Staubli VAL3: JTrajPtFullBody.dtx

public num accelerations[10]
public num positions[10]
public num robotId
public num sequence
public num time
public num validFields
public num velocities[10]
